INTERFACE I_FieldDevice

METHOD M_DeviceEnable : BOOL
VAR_INPUT
END_VAR
END_METHOD

METHOD M_DeviceHeartbeat : BOOL
VAR_INPUT
END_VAR
END_METHOD

METHOD M_DeviceReset : BOOL
VAR_INPUT
END_VAR
END_METHOD

METHOD M_DeviceStatus : E_StatusFieldDevice
VAR_INPUT
END_VAR
END_METHOD

PROPERTY pDeviceCommOK : BOOL
GET
END_GET
SET
END_SET
END_PROPERTY

PROPERTY pDeviceEnableCmd : BOOL
GET
END_GET
SET
END_SET
END_PROPERTY

PROPERTY pDeviceEnabled : BOOL
GET
END_GET
SET
END_SET
END_PROPERTY

PROPERTY pDeviceFaulted : BOOL
GET
END_GET
SET
END_SET
END_PROPERTY

PROPERTY pDeviceReset : BOOL
SET
END_SET
END_PROPERTY

PROPERTY pDeviceStatusFeedback : DWORD
GET
END_GET
SET
END_SET
END_PROPERTY

END_INTERFACE

(* stored: Version 1.1.0.1, ProductVersion 3.1.4024.15
   Itf I_FieldDevice: Id {da4e5490-5768-4d44-b47a-f8648bda148f}
   Method M_DeviceEnable: Id {66611878-468d-4a93-abc8-e579085825ea}
   Method M_DeviceHeartbeat: Id {d929bca2-a963-4538-b506-159be56dca41}
   Method M_DeviceReset: Id {28520df0-2b3b-4670-8924-aeb864750682}
   Method M_DeviceStatus: Id {78fe631b-ed6a-4e93-bc55-568c4437fab0}
   Property pDeviceCommOK: Id {32dd4ea4-a3ba-4192-bdcb-500e51e37f04}
   Get Get: Id {209928c4-65f1-4fae-8525-50042034e99b}
   Set Set: Id {12f53733-64ab-4dee-9ef0-6a3ad19c5112}
   Property pDeviceEnableCmd: Id {11802a59-9ca7-46cc-9f43-e70f3ab25899}
   Get Get: Id {60ce9367-e3c7-4c41-877e-7efe8ddc638d}
   Set Set: Id {8f13aa7f-877e-41bd-82d5-85e3916fc299}
   Property pDeviceEnabled: Id {018891a8-c2f0-4797-b63a-0043f5a77bef}
   Get Get: Id {3617add4-7ddd-4c17-bdea-8934921f9e34}
   Set Set: Id {1f83d461-0914-4c80-be17-2d5e4625ef73}
   Property pDeviceFaulted: Id {f7358a9d-1711-4995-bebd-56e2b259beb1}
   Get Get: Id {cac6c2a6-8361-4327-918c-25408f44224b}
   Set Set: Id {9445234f-6a17-46a2-9b5a-6b61063cb6a1}
   Property pDeviceReset: Id {8ffe5666-d627-4cc2-978b-bb0403f28d7a}
   Set Set: Id {c6befaf6-e2df-44c0-aaff-c3d90284af41}
   Property pDeviceStatusFeedback: Id {950e1948-37c0-43fb-8757-34f5b6791a86}
   Get Get: Id {63d31bd8-0eb5-49e1-af1f-6998abc8c831}
   Set Set: Id {e2193345-8e14-41b7-a413-da901e6fa7c7} *)
